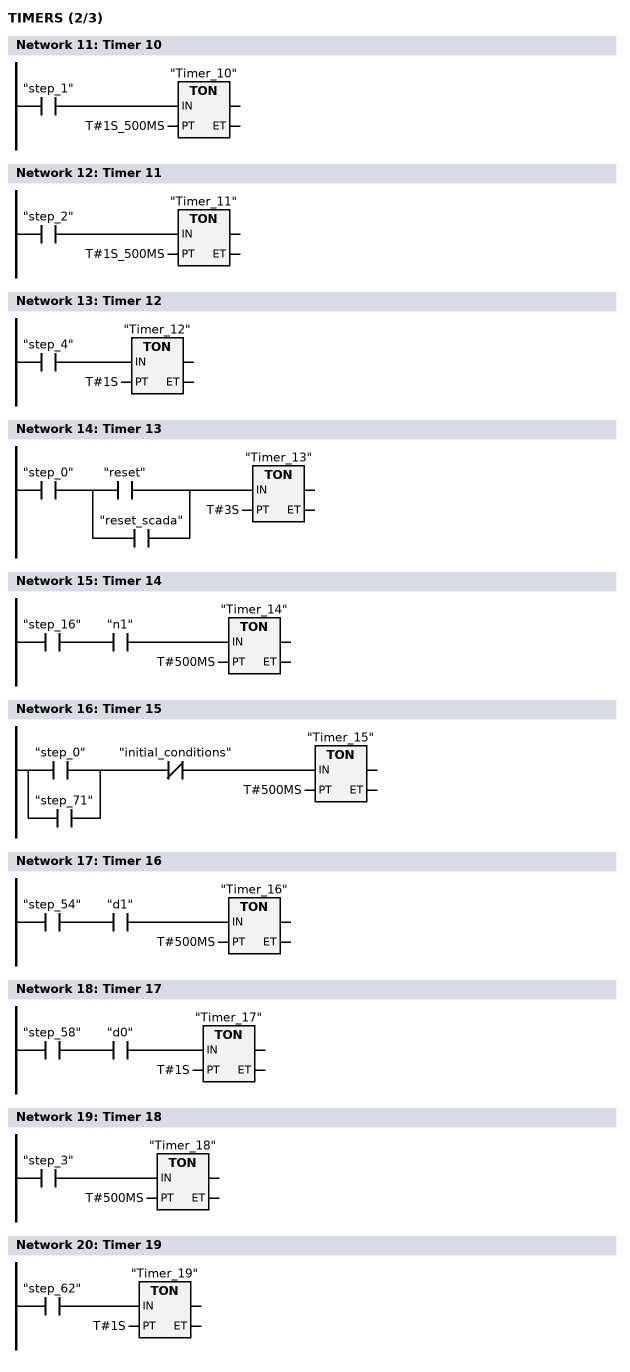
   "Timer_10".TON(IN := "step_1", PT := T#1S_500MS);
END_REGION

REGION Network 12: Timer 11
   "Timer_11".TON(IN := "step_2", PT := T#1S_500MS);
END_REGION

REGION Network 13: Timer 12
   "Timer_12".TON(IN := "step_4", PT := T#1S);
END_REGION

REGION Network 14: Timer 13
   "Timer_13".TON(IN := "step_0" AND ("reset" OR "reset_scada"), PT := T#3S);
END_REGION

REGION Network 15: Timer 14
   "Timer_14".TON(IN := "step_16" AND "n1", PT := T#500MS);
END_REGION

REGION Network 16: Timer 15
   "Timer_15".TON(IN := ("step_0" OR "step_71") AND NOT "initial_conditions", PT := T#500MS);
END_REGION

REGION Network 17: Timer 16
   "Timer_16".TON(IN := "step_54" AND "d1", PT := T#500MS);
END_REGION

REGION Network 18: Timer 17
   "Timer_17".TON(IN := "step_58" AND "d0", PT := T#1S);
END_REGION

REGION Network 19: Timer 18
   "Timer_18".TON(IN := "step_3", PT := T#500MS);
END_REGION

REGION Network 20: Timer 19
   "Timer_19".TON(IN := "step_62", PT := T#1S);
END_REGION

REGION Network 21: Timer 20
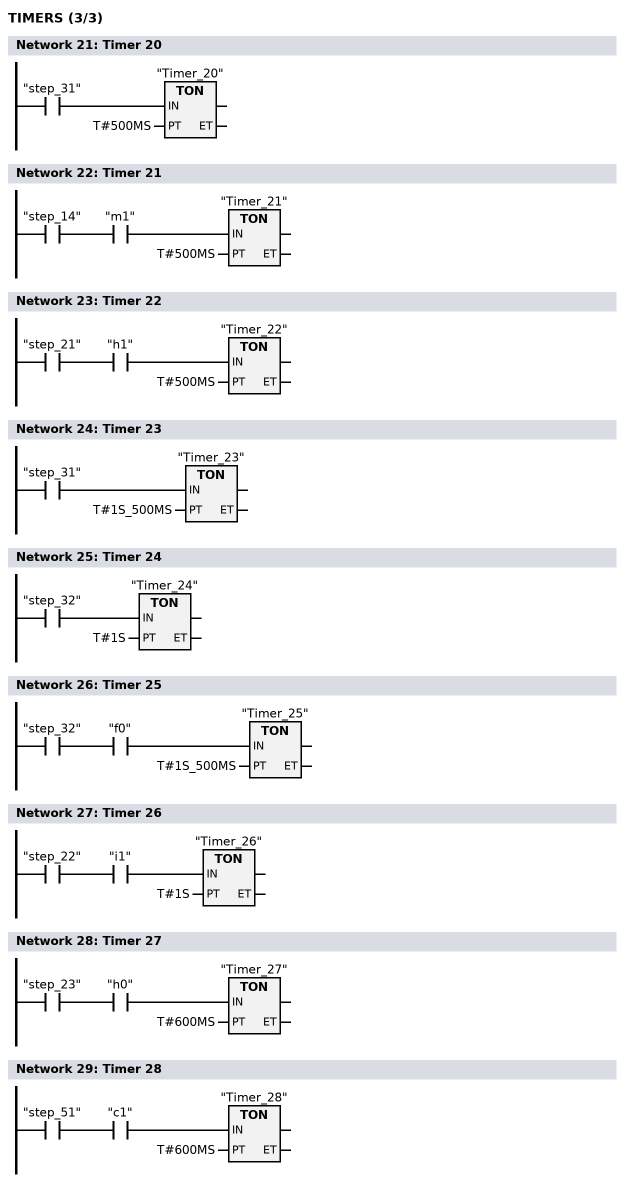
   "Timer_20".TON(IN := "step_31", PT := T#500MS);
END_REGION

REGION Network 22: Timer 21
   "Timer_21".TON(IN := "step_14" AND "m1", PT := T#500MS);
END_REGION

REGION Network 23: Timer 22
   "Timer_22".TON(IN := "step_21" AND "h1", PT := T#500MS);
END_REGION

REGION Network 24: Timer 23
   "Timer_23".TON(IN := "step_31", PT := T#1S_500MS);
END_REGION

REGION Network 25: Timer 24
   "Timer_24".TON(IN := "step_32", PT := T#1S);
END_REGION

REGION Network 26: Timer 25
   "Timer_25".TON(IN := "step_32" AND "f0", PT := T#1S_500MS);
END_REGION

REGION Network 27: Timer 26
   "Timer_26".TON(IN := "step_22" AND "i1", PT := T#1S);
END_REGION

REGION Network 28: Timer 27
   "Timer_27".TON(IN := "step_23" AND "h0", PT := T#600MS);
END_REGION

REGION Network 29: Timer 28
   "Timer_28".TON(IN := "step_51" AND "c1", PT := T#600MS);
END_REGION
END_FUNCTION

FUNCTION "OUTPUTS" : Void   // FC4, LAD
TITLE = OUTPUTS
{ S7_Optimized_Access := 'TRUE' }
VERSION : 0.1
BEGIN

REGION Network 1: Red light
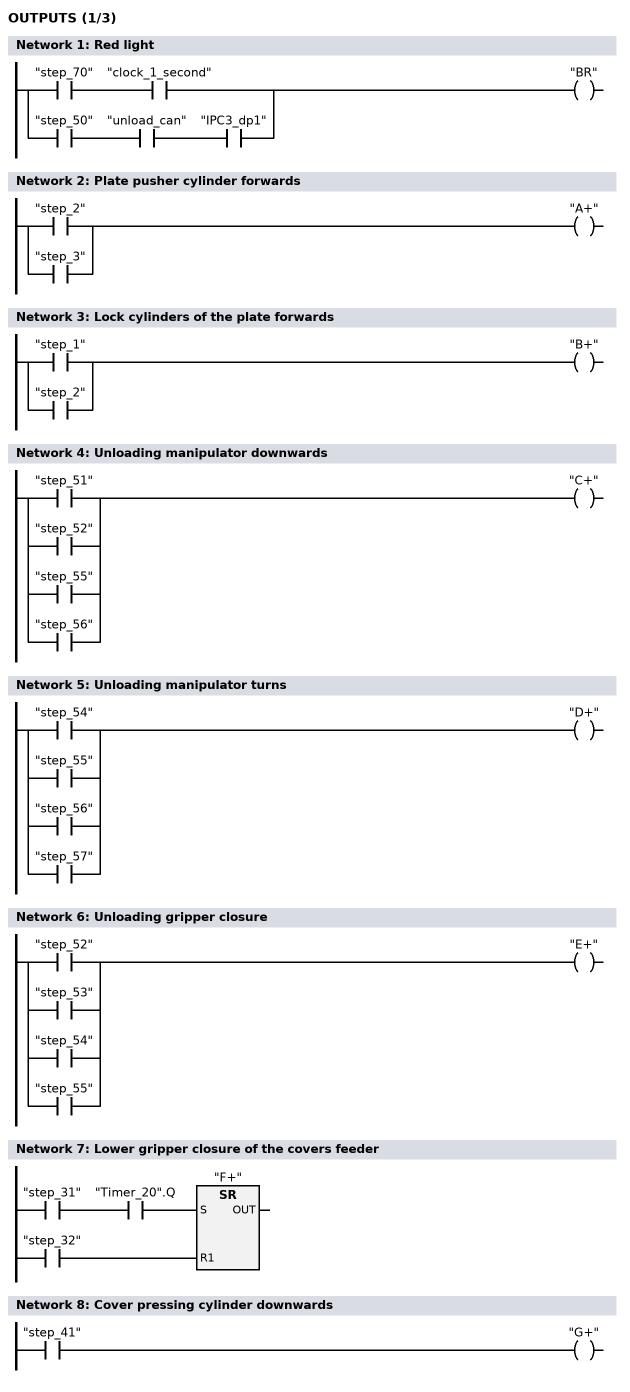
   RUNG wire#powerrail
      Contact( "step_70" )
      Contact( "clock_1_second" )
      wire#w1
      Coil( "BR" )
   END_RUNG
   RUNG wire#powerrail
      Contact( "step_50" )
      Contact( "unload_can" )
      Contact( "IPC3_dp1" )
   END_RUNG wire#w1
   // the same network as SCL:
   "BR" := ("step_70" AND "clock_1_second") OR ("step_50" AND "unload_can" AND "IPC3_dp1");
END_REGION

REGION Network 2: Plate pusher cylinder forwards
   RUNG wire#powerrail
      Contact( "step_2" )
      wire#w1
      Coil( "A+" )
   END_RUNG
   RUNG wire#powerrail
      Contact( "step_3" )
   END_RUNG wire#w1
   // the same network as SCL:
   "A+" := "step_2" OR "step_3";
END_REGION

REGION Network 3: Lock cylinders of the plate forwards
   RUNG wire#powerrail
      Contact( "step_1" )
      wire#w1
      Coil( "B+" )
   END_RUNG
   RUNG wire#powerrail
      Contact( "step_2" )
   END_RUNG wire#w1
   // the same network as SCL:
   "B+" := "step_1" OR "step_2";
END_REGION

REGION Network 4: Unloading manipulator downwards
   RUNG wire#powerrail
      Contact( "step_51" )
      wire#w1
      Coil( "C+" )
   END_RUNG
   RUNG wire#powerrail
      Contact( "step_52" )
   END_RUNG wire#w1
   RUNG wire#powerrail
      Contact( "step_55" )
   END_RUNG wire#w1
   RUNG wire#powerrail
      Contact( "step_56" )
   END_RUNG wire#w1
   // the same network as SCL:
   "C+" := "step_51" OR "step_52" OR "step_55" OR "step_56";
END_REGION

REGION Network 5: Unloading manipulator turns
   RUNG wire#powerrail
      Contact( "step_54" )
      wire#w1
      Coil( "D+" )
   END_RUNG
   RUNG wire#powerrail
      Contact( "step_55" )
   END_RUNG wire#w1
   RUNG wire#powerrail
      Contact( "step_56" )
   END_RUNG wire#w1
   RUNG wire#powerrail
      Contact( "step_57" )
   END_RUNG wire#w1
   // the same network as SCL:
   "D+" := "step_54" OR "step_55" OR "step_56" OR "step_57";
END_REGION

REGION Network 6: Unloading gripper closure
   RUNG wire#powerrail
      Contact( "step_52" )
      wire#w1
      Coil( "E+" )
   END_RUNG
   RUNG wire#powerrail
      Contact( "step_53" )
   END_RUNG wire#w1
   RUNG wire#powerrail
      Contact( "step_54" )
   END_RUNG wire#w1
   RUNG wire#powerrail
      Contact( "step_55" )
   END_RUNG wire#w1
   // the same network as SCL:
   "E+" := "step_52" OR "step_53" OR "step_54" OR "step_55";
END_REGION

REGION Network 7: Lower gripper closure of the covers feeder
   RUNG wire#powerrail
      Contact( "step_31" )
      Contact( "Timer_20".Q )
      S_SR(operand := "F+", r1 := wire#w1)
   END_RUNG
   RUNG wire#powerrail
      Contact( "step_32" )
   END_RUNG wire#w1
   // the same network as SCL:
   IF "step_31" AND "Timer_20".Q THEN
       "F+" := TRUE;   // SR flip-flop
   END_IF;
   IF "step_32" THEN "F+" := FALSE; END_IF;
END_REGION

REGION Network 8: Cover pressing cylinder downwards
   RUNG wire#powerrail
      Contact( "step_41" )
      Coil( "G+" )
   END_RUNG
   // the same network as SCL:
   "G+" := "step_41";
END_REGION

REGION Network 9: Load manipulator upwards
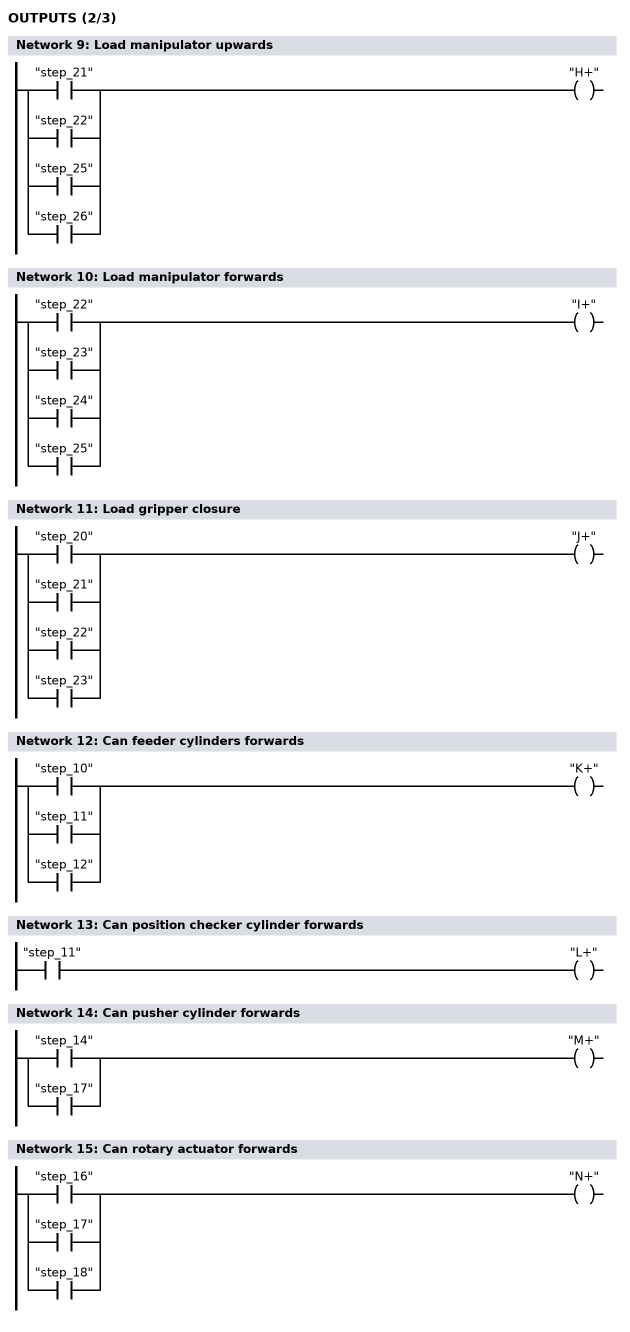
   RUNG wire#powerrail
      Contact( "step_21" )
      wire#w1
      Coil( "H+" )
   END_RUNG
   RUNG wire#powerrail
      Contact( "step_22" )
   END_RUNG wire#w1
   RUNG wire#powerrail
      Contact( "step_25" )
   END_RUNG wire#w1
   RUNG wire#powerrail
      Contact( "step_26" )
   END_RUNG wire#w1
   // the same network as SCL:
   "H+" := "step_21" OR "step_22" OR "step_25" OR "step_26";
END_REGION

REGION Network 10: Load manipulator forwards
   RUNG wire#powerrail
      Contact( "step_22" )
      wire#w1
      Coil( "I+" )
   END_RUNG
   RUNG wire#powerrail
      Contact( "step_23" )
   END_RUNG wire#w1
   RUNG wire#powerrail
      Contact( "step_24" )
   END_RUNG wire#w1
   RUNG wire#powerrail
      Contact( "step_25" )
   END_RUNG wire#w1
   // the same network as SCL:
   "I+" := "step_22" OR "step_23" OR "step_24" OR "step_25";
END_REGION

REGION Network 11: Load gripper closure
   RUNG wire#powerrail
      Contact( "step_20" )
      wire#w1
      Coil( "J+" )
   END_RUNG
   RUNG wire#powerrail
      Contact( "step_21" )
   END_RUNG wire#w1
   RUNG wire#powerrail
      Contact( "step_22" )
   END_RUNG wire#w1
   RUNG wire#powerrail
      Contact( "step_23" )
   END_RUNG wire#w1
   // the same network as SCL:
   "J+" := "step_20" OR "step_21" OR "step_22" OR "step_23";
END_REGION

REGION Network 12: Can feeder cylinders forwards
   RUNG wire#powerrail
      Contact( "step_10" )
      wire#w1
      Coil( "K+" )
   END_RUNG
   RUNG wire#powerrail
      Contact( "step_11" )
   END_RUNG wire#w1
   RUNG wire#powerrail
      Contact( "step_12" )
   END_RUNG wire#w1
   // the same network as SCL:
   "K+" := "step_10" OR "step_11" OR "step_12";
END_REGION

REGION Network 13: Can position checker cylinder forwards
   RUNG wire#powerrail
      Contact( "step_11" )
      Coil( "L+" )
   END_RUNG
   // the same network as SCL:
   "L+" := "step_11";
END_REGION

REGION Network 14: Can pusher cylinder forwards
   RUNG wire#powerrail
      Contact( "step_14" )
      wire#w1
      Coil( "M+" )
   END_RUNG
   RUNG wire#powerrail
      Contact( "step_17" )
   END_RUNG wire#w1
   // the same network as SCL:
   "M+" := "step_14" OR "step_17";
END_REGION

REGION Network 15: Can rotary actuator forwards
   RUNG wire#powerrail
      Contact( "step_16" )
      wire#w1
      Coil( "N+" )
   END_RUNG
   RUNG wire#powerrail
      Contact( "step_17" )
   END_RUNG wire#w1
   RUNG wire#powerrail
      Contact( "step_18" )
   END_RUNG wire#w1
   // the same network as SCL:
   "N+" := "step_16" OR "step_17" OR "step_18";
END_REGION

REGION Network 16: Upper gripper closure of the covers feeder
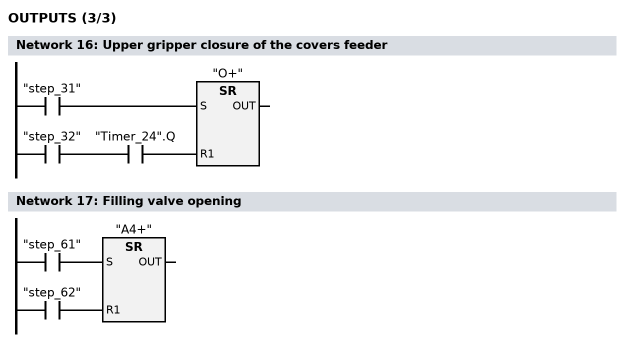
   RUNG wire#powerrail
      Contact( "step_31" )
      S_SR(operand := "O+", r1 := wire#w1)
   END_RUNG
   RUNG wire#powerrail
      Contact( "step_32" )
      Contact( "Timer_24".Q )
   END_RUNG wire#w1
   // the same network as SCL:
   IF "step_31" THEN
       "O+" := TRUE;   // SR flip-flop
   END_IF;
   IF "step_32" AND "Timer_24".Q THEN "O+" := FALSE; END_IF;
END_REGION

REGION Network 17: Filling valve opening
   RUNG wire#powerrail
      Contact( "step_61" )
      S_SR(operand := "A4+", r1 := wire#w1)
   END_RUNG
   RUNG wire#powerrail
      Contact( "step_62" )
   END_RUNG wire#w1
   // the same network as SCL:
   IF "step_61" THEN
       "A4+" := TRUE;   // SR flip-flop
   END_IF;
   IF "step_62" THEN "A4+" := FALSE; END_IF;
END_REGION
END_FUNCTION

FUNCTION "COMMUNICATIONS" : Void   // FC5, LAD
TITLE = COMMUNICATIONS
{ S7_Optimized_Access := 'TRUE' }
VERSION : 0.1
BEGIN

REGION Network 1: GET function (reading from IPC201C)
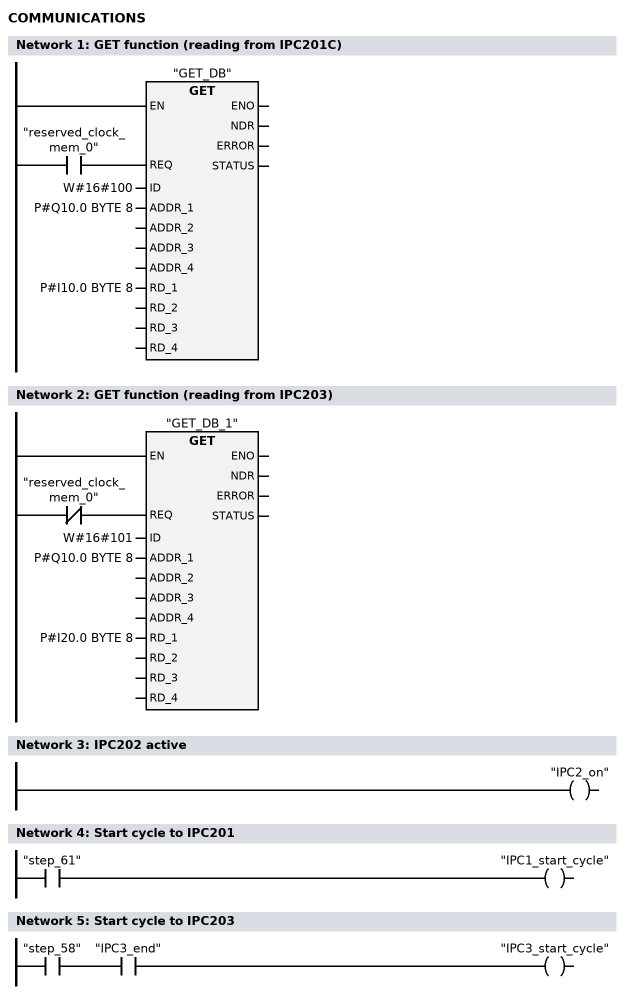
   "GET_DB"(REQ := "reserved_clock_mem_0", ID := W#16#100, ADDR_1 := P#Q10.0 BYTE 8, RD_1 := P#I10.0 BYTE 8);   // GET
END_REGION

REGION Network 2: GET function (reading from IPC203)
   "GET_DB_1"(REQ := NOT "reserved_clock_mem_0",   // GET
              ID := W#16#101,
              ADDR_1 := P#Q10.0 BYTE 8,
              RD_1 := P#I20.0 BYTE 8);
END_REGION

REGION Network 3: IPC202 active
   RUNG wire#powerrail
      Coil( "IPC2_on" )
   END_RUNG
   // the same network as SCL:
   "IPC2_on" := TRUE;
END_REGION

REGION Network 4: Start cycle to IPC201
   RUNG wire#powerrail
      Contact( "step_61" )
      Coil( "IPC1_start_cycle" )
   END_RUNG
   // the same network as SCL:
   "IPC1_start_cycle" := "step_61";
END_REGION

REGION Network 5: Start cycle to IPC203
   RUNG wire#powerrail
      Contact( "step_58" )
      Contact( "IPC3_end" )
      Coil( "IPC3_start_cycle" )
   END_RUNG
   // the same network as SCL:
   "IPC3_start_cycle" := "step_58" AND "IPC3_end";
END_REGION
END_FUNCTION

FUNCTION "SCADA" : Void   // FC6, LAD
TITLE = SCADA
{ S7_Optimized_Access := 'TRUE' }
VERSION : 0.1
BEGIN

REGION Network 1: Output channel 0 to SCADA
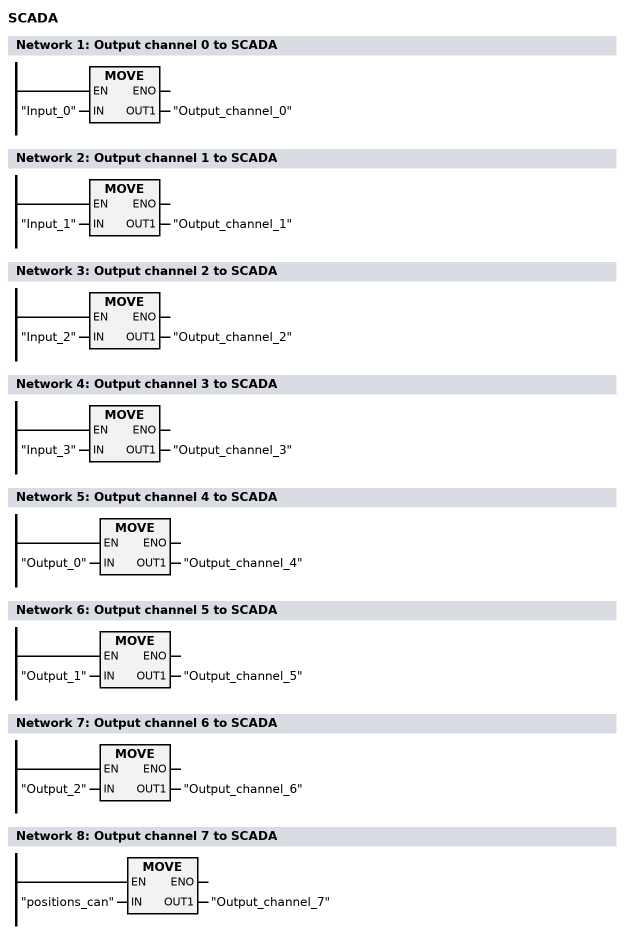
   RUNG wire#powerrail
      { S7_GenerateENO := "TRUE" } Move(in := "Input_0", out1 => "Output_channel_0")
   END_RUNG
   // the same network as SCL:
   "Output_channel_0" := "Input_0";
END_REGION

REGION Network 2: Output channel 1 to SCADA
   RUNG wire#powerrail
      { S7_GenerateENO := "TRUE" } Move(in := "Input_1", out1 => "Output_channel_1")
   END_RUNG
   // the same network as SCL:
   "Output_channel_1" := "Input_1";
END_REGION

REGION Network 3: Output channel 2 to SCADA
   RUNG wire#powerrail
      { S7_GenerateENO := "TRUE" } Move(in := "Input_2", out1 => "Output_channel_2")
   END_RUNG
   // the same network as SCL:
   "Output_channel_2" := "Input_2";
END_REGION

REGION Network 4: Output channel 3 to SCADA
   RUNG wire#powerrail
      { S7_GenerateENO := "TRUE" } Move(in := "Input_3", out1 => "Output_channel_3")
   END_RUNG
   // the same network as SCL:
   "Output_channel_3" := "Input_3";
END_REGION

REGION Network 5: Output channel 4 to SCADA
   RUNG wire#powerrail
      { S7_GenerateENO := "TRUE" } Move(in := "Output_0", out1 => "Output_channel_4")
   END_RUNG
   // the same network as SCL:
   "Output_channel_4" := "Output_0";
END_REGION

REGION Network 6: Output channel 5 to SCADA
   RUNG wire#powerrail
      { S7_GenerateENO := "TRUE" } Move(in := "Output_1", out1 => "Output_channel_5")
   END_RUNG
   // the same network as SCL:
   "Output_channel_5" := "Output_1";
END_REGION

REGION Network 7: Output channel 6 to SCADA
   RUNG wire#powerrail
      { S7_GenerateENO := "TRUE" } Move(in := "Output_2", out1 => "Output_channel_6")
   END_RUNG
   // the same network as SCL:
   "Output_channel_6" := "Output_2";
END_REGION

REGION Network 8: Output channel 7 to SCADA
   RUNG wire#powerrail
      { S7_GenerateENO := "TRUE" } Move(in := "positions_can", out1 => "Output_channel_7")
   END_RUNG
   // the same network as SCL:
   "Output_channel_7" := "positions_can";
END_REGION
END_FUNCTION

ORGANIZATION_BLOCK "Main"   // OB1, LAD, ProgramCycle
TITLE = "Main Program Sweep (Cycle)"
{ S7_Optimized_Access := 'TRUE' }
VERSION : 0.1
   VAR_INPUT
      Initial_Call : Bool;   // Initial call of this OB
      Remanence : Bool;   // =True, if remanent data are available
   END_VAR
BEGIN

REGION Network 1: Call to STEPS routine
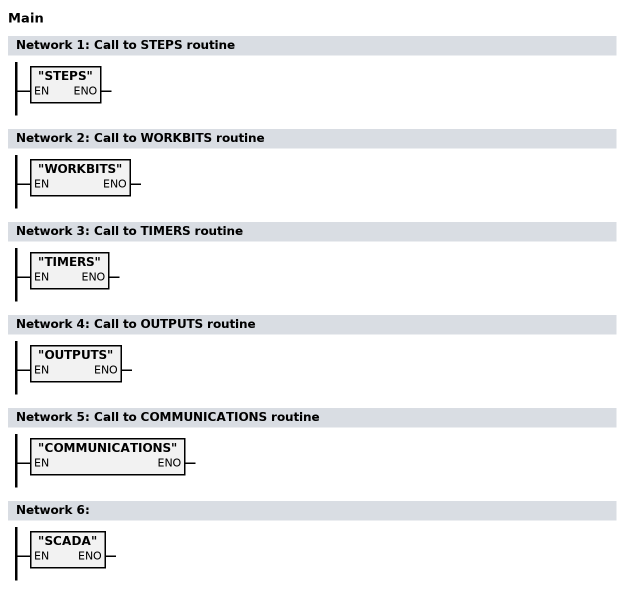
   RUNG wire#powerrail
      "STEPS"()
   END_RUNG
   // the same network as SCL:
   "STEPS"();
END_REGION

REGION Network 2: Call to WORKBITS routine
   RUNG wire#powerrail
      "WORKBITS"()
   END_RUNG
   // the same network as SCL:
   "WORKBITS"();
END_REGION

REGION Network 3: Call to TIMERS routine
   RUNG wire#powerrail
      "TIMERS"()
   END_RUNG
   // the same network as SCL:
   "TIMERS"();
END_REGION

REGION Network 4: Call to OUTPUTS routine
   RUNG wire#powerrail
      "OUTPUTS"()
   END_RUNG
   // the same network as SCL:
   "OUTPUTS"();
END_REGION

REGION Network 5: Call to COMMUNICATIONS routine
   RUNG wire#powerrail
      "COMMUNICATIONS"()
   END_RUNG
   // the same network as SCL:
   "COMMUNICATIONS"();
END_REGION

REGION Network 6
   RUNG wire#powerrail
      "SCADA"()
   END_RUNG
   // the same network as SCL:
   "SCADA"();
END_REGION
END_ORGANIZATION_BLOCK

ORGANIZATION_BLOCK "Startup"   // OB100, LAD, Startup
TITLE = "Complete Restart"
{ S7_Optimized_Access := 'TRUE' }
VERSION : 0.1
   VAR_INPUT
      LostRetentive : Bool;   // True if retentive data are lost
      LostRTC : Bool;   // True if date and time are lost
   END_VAR
BEGIN

REGION Network 1: Activation of the first step of the Grafcet (Step 0)
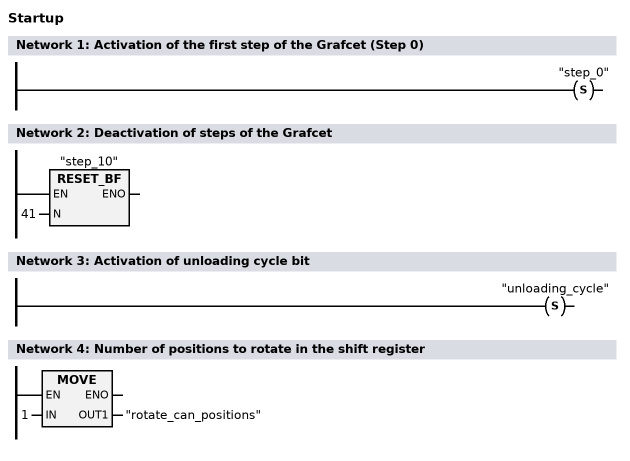
   RUNG wire#powerrail
      S_Coil( "step_0" )
   END_RUNG
   // the same network as SCL:
   "step_0" := TRUE;
END_REGION

REGION Network 2: Deactivation of steps of the Grafcet
   // no SCL statement known for RBitfield: written as a call
   RESET_BF(operand := "step_10", n := 41);
END_REGION

REGION Network 3: Activation of unloading cycle bit
   RUNG wire#powerrail
      S_Coil( "unloading_cycle" )
   END_RUNG
   // the same network as SCL:
   "unloading_cycle" := TRUE;
END_REGION

REGION Network 4: Number of positions to rotate in the shift register
   RUNG wire#powerrail
      Move(in := 1, out1 => "rotate_can_positions")
   END_RUNG
   // the same network as SCL:
   "rotate_can_positions" := 1;
END_REGION
END_ORGANIZATION_BLOCK

// ===== PLC "PLC_1"  CPU 1214C DC/DC/DC =====

ORGANIZATION_BLOCK "Main"   // OB1, LAD, ProgramCycle
TITLE = "Main Program Sweep (Cycle)"
{ S7_Optimized_Access := 'TRUE' }
VERSION : 0.1
   VAR_INPUT
      Initial_Call : Bool;   // Initial call of this OB
      Remanence : Bool;   // =True, if remanent data are available
   END_VAR
BEGIN
END_ORGANIZATION_BLOCK